{attribute 'qualified_only'}
VAR_GLOBAL
strActiveMastersList:ARRAY[1..etherCATdiag.maxNumEtherCATmasters] OF STRING(23);	
valActiveMastersSel:UDINT;
END_VAR

(* stored: Version 1.1.0.1, ProductVersion 3.1.4024.12
   GVL etherCATmasters: Id {ab5f070f-5140-43fa-8291-68b78e1c7fbc} *)
